TYPE AX5000_S_0024 :
STRUCT
	Actual_lenght:UINT;
	Max_lenght:UINT;
	Configuration_list_of_MDT:ARRAY[0..11] OF UINT;
END_STRUCT
END_TYPE

(* stored: Version 1.1.0.1, ProductVersion 3.1.4024.3
   DUT AX5000_S_0024: Id {ebc8fbc6-d47e-4eb8-8042-dad8ebaf09af} *)
